FUNCTION_BLOCK EL3051
VAR
	_io : EL3xx1_Data;
	{attribute addProperty Name "WcState"}
	_wcState : WcStateInputToggle;
	{attribute addProperty Name "Info data"}
	_infoData : InfoDataAds;
END_VAR

PROPERTY IO : REFERENCE TO EL3xx1_Data
GET
IO REF= _io;
END_GET
END_PROPERTY

PROPERTY WcState : REFERENCE TO WcStateInputToggle
GET
WcState REF= _wcState;
END_GET
END_PROPERTY

END_FUNCTION_BLOCK

(* stored: Version 1.1.0.1, ProductVersion 3.1.4024.9
   POU EL3051: Id {10dd2dce-16e9-0375-2373-2a1054afb3ed}, SpecialFunc None
   Property IO: Id {ff6cce23-b690-0418-0542-99c035c1e5b9}
   Get Get: Id {c3f7a1a4-e465-0dda-2d93-af6a314f1d6d}
   Property WcState: Id {1932c050-a0dc-07e5-1ccb-0fe793591971}
   Get Get: Id {11dd2a79-6d90-0526-3eb2-f929c0bff88b} *)
